FOR K2:=0 TO 5 DO
	 Cn_date[20,K2]:=0;
	 Cn_date[21,K2]:=0;
	 Cn_date[22,K2]:=0;
	 Cn_date[23,K2]:=0;
	 Cn_date[0,K2]:=0;
	 Cn_date[1,K2]:=0;
	 Cn_date[2,K2]:=0;
	 Cn_date[3,K2]:=0;
	 Cn_date[4,K2]:=0;
	 Cn_date[5,K2]:=0;
	 Cn_date[6,K2]:=0;
	 Cn_date[7,K2]:=0;
END_FOR
NGMark2[0,0]:=0;
NGMark2[1,0]:=0;
NGMark2[2,0]:=0;
NGMark2[3,0]:=0;
NGMark2[4,0]:=0;
NGMark2[5,0]:=0;
NGMark2[6,0]:=0;
NGMark2[7,0]:=0;
NGMark2[8,0]:=0;
NGMark2[9,0]:=0;
NGMark2[10,0]:=0;
NGMark2[11,0]:=0;
NGMark2[12,0]:=0;
NGMark2[13,0]:=0;
NGMark2[14,0]:=0;
NGMark2[0,0]:=0;
NGMark2[1,1]:=0;
NGMark2[2,1]:=0;
NGMark2[3,1]:=0;
NGMark2[4,1]:=0;
NGMark2[5,1]:=0;
NGMark2[6,1]:=0;
NGMark2[7,1]:=0;
NGMark2[8,1]:=0;
NGMark2[9,1]:=0;
NGMark2[10,1]:=0;
NGMark2[11,1]:=0;
NGMark2[12,1]:=0;
NGMark2[13,1]:=0;
NGMark2[14,1]:=0;
END_IF

END_FUNCTION_BLOCK

// ---- POUs/BasicFunction/Data/FB_DataTime.TcPOU
FUNCTION_BLOCK FB_DataTime
VAR_INPUT
	Month:INT;//实时月；
	dDay:INT;//实时日期；
	Hour:INT;//当前时间小时；
	Mins:INT;//分钟；
   Second:INT;//秒
    Alm :    BOOL ;//报警
	Wait :BOOL ;//待机
	Run :BOOL ;//运行
	JP_Wait:BOOL ;//极片更换时间
	Query:BOOL;//时间查询
	

END_VAR
VAR_OUTPUT
		STTimedata:ARRAY[0..32] OF ST_Timedata_2;

END_VAR
VAR
	
	rRun : R_TRIG;
	rAlm : R_TRIG;
	rWait : R_TRIG;
	rXL_Wait : R_TRIG;
	
	fRun: F_TRIG;
	fAlm: F_TRIG;
	fWait: F_TRIG;
    delay:BOOL ;//延时
	TON_1: TON;
	i:INT;
	K: INT;
	J: BOOL;
END_VAR

VAR_IN_OUT
     date1:INT;//查询日期
END_VAR

K:=K+1;
	IF K>499THEN
		J:=TRUE;
		K:=0;
	ELSE
		J:=FALSE;
	END_IF




///////////////运行时间/////////////////
rRun(CLK:= J , Q=> );

IF rRun.Q  AND  Run THEN
	STTimedata[System.StTime.wDay].RunTime[System.StTime.wHour]:=STTimedata[System.StTime.wDay].RunTime[System.StTime.wHour]+1;
END_IF

IF STTimedata[System.StTime.wDay].RunTime[System.StTime.wHour]> 3600 THEN
	STTimedata[System.StTime.wDay].RunTime[System.StTime.wHour]:= 3600 ;
END_IF

//IF STTimedata[System.StTime.wDay].AlmTime[System.StTime.wHour]= 0 AND STTimedata[System.StTime.wDay].WaitTime[System.StTime.wHour]= 0  AND 
 //   (STTimedata[System.StTime.wDay].RunTime[System.StTime.wHour]= 3585  OR  STTimedata[System.StTime.wDay].RunTime[System.StTime.wHour]= 3586 ) THEN
	//STTimedata[System.StTime.wDay].RunTime[System.StTime.wHour]:= 3600 ;
//END_IF


///////////////待机时间///////////////
rWait(CLK:=J , Q=> );

IF rWait.Q  AND Wait THEN
	STTimedata[System.StTime.wDay].WaitTime[System.StTime.wHour]:=STTimedata[System.StTime.wDay].WaitTime[System.StTime.wHour]+1;
END_IF

IF STTimedata[System.StTime.wDay].WaitTime[System.StTime.wHour]> 3600 THEN
	STTimedata[System.StTime.wDay].WaitTime[System.StTime.wHour]:= 3600 ;
END_IF

//IF STTimedata[System.StTime.wDay].RunTime[System.StTime.wHour]= 0 AND STTimedata[System.StTime.wDay].AlmTime[System.StTime.wHour]= 0  AND 
  //   (STTimedata[System.StTime.wDay].RunTime[System.StTime.wHour]= 3585  OR  STTimedata[System.StTime.wDay].RunTime[System.StTime.wHour]= 3586 )  THEN
//	STTimedata[System.StTime.wDay].WaitTime[System.StTime.wHour]:= 3600 ;
//END_IF


////////////////报警时间///////////////
rAlm(CLK:=J , Q=> );

IF rAlm.Q AND Alm THEN
	STTimedata[System.StTime.wDay].AlmTime[System.StTime.wHour]:=STTimedata[System.StTime.wDay].AlmTime[System.StTime.wHour]+1;
END_IF

IF STTimedata[System.StTime.wDay].AlmTime[System.StTime.wHour]> 3600 THEN
	STTimedata[System.StTime.wDay].AlmTime[System.StTime.wHour]:= 3600 ;
END_IF

//IF STTimedata[System.StTime.wDay].RunTime[System.StTime.wHour]= 0 AND STTimedata[System.StTime.wDay].WaitTime[System.StTime.wHour]= 0  AND
//    (STTimedata[System.StTime.wDay].RunTime[System.StTime.wHour]= 3585  OR  STTimedata[System.StTime.wDay].RunTime[System.StTime.wHour]= 3586 ) THEN
//	STTimedata[System.StTime.wDay].AlmTime[System.StTime.wHour]:= 3600 ;
//END_IF

////////////////下料等待托盘时间///////////////
rXL_Wait(CLK:=J, Q=> );

IF rXL_Wait.Q AND JP_Wait THEN
	STTimedata[System.StTime.wDay].changeTime[System.StTime.wHour]:=STTimedata[System.StTime.wDay].changeTime[System.StTime.wHour]+1;
END_IF

//数据查询
IF Query THEN
	delay:=TRUE;
END_IF

TON_1(IN:= , PT:=T#60S , Q=> , ET=> );
IF delay THEN
		  IF NOT TON_1.Q THEN
			  TON_1.IN:=TRUE;
		  ELSE	
			  delay:=FALSE;
			  date1:=System.StTime.wDay;
		  END_IF	 
ELSE	
	 TON_1.IN:=FALSE;
END_IF


IF NOT delay THEN
STTimedata[32]:=STTimedata[System.StTime.wDay];
ELSE
STTimedata[32]:=STTimedata[date1];
END_IF

//数据清零
IF (System.StTime.wMonth=2 AND  System.StTime.wDay=28 )   OR
    ((System.StTime.wMonth=4 OR System.StTime.wMonth=6 OR System.StTime.wMonth=9 OR System.StTime.wMonth=11) AND System.StTime.wDay=30 )   OR
	((System.StTime.wMonth=1 OR  System.StTime.wMonth=3 OR System.StTime.wMonth=5 OR System.StTime.wMonth=7 OR System.StTime.wMonth=8 OR System.StTime.wMonth=10 OR System.StTime.wMonth=12) AND  System.StTime.wDay=31)  AND
    System.StTime.wHour=23 AND   System.StTime.wMinute =59 AND  System.StTime.wSecond =59 THEN
	FOR i:=0 TO 32  DO
	MEMSET(ADR(STTimedata[i]),0,SIZEOF(STTimedata[i]));	
	END_FOR
END_IF

END_FUNCTION_BLOCK

// ---- POUs/BasicFunction/Data/CS_Recipe.TcPOU
FUNCTION_BLOCK CS_Recipe
VAR_INPUT
END_VAR
VAR_OUTPUT
END_VAR
VAR
	


 //recipeManCommands: RecipeManCommands;
	result: DWORD;
END_VAR

VAR_IN_OUT
  iRecipe2:    IRecipe;
END_VAR





(*

IF iRecipe2.bCreate THEN
   result:= recipeManCommands.CreateRecipe(RecipeDefinitionName:='Recipes' , RecipeName:='SJ_Rec' );
   iRecipe2.bCreate:=FALSE;
END_IF

IF iRecipe2.bSave THEN
    result:= recipeManCommands.ReadAndSaveRecipeAs(RecipeDefinitionName:='Recipes' , RecipeName:='SJ_Rec' , FileName:='C:\P2Data\P2Par');
    iRecipe2.bSave:=FALSE;
END_IF

IF iRecipe2.bLoad THEN
	result:= RecipeManCommands.LoadFromAndWriteRecipe(RecipeDefinitionName:='Recipes' , RecipeName:='SJ_Rec' , FileName:='C:\P2Data\P2Par');
    iRecipe2.bLoad:=FALSE;
END_IF

*)

END_FUNCTION_BLOCK

// ---- POUs/BasicFunction/MES/CS_CcdTcp_V2.TcPOU
FUNCTION_BLOCK PUBLIC CS_CcdTcp_V2
VAR_INPUT
END_VAR
VAR_OUTPUT
END_VAR
VAR_IN_OUT
   iCcd2:ST_CCDCom;
   Data:STCcdData;
END_VAR


VAR
	ccdDataSend:STCcdDataSend;
	ccdDataReceive:STCcdDataSend;
	fbTcpCon:FB_SocketConnect;
	fbTcpSend:FB_SocketSend;
	fbTcpRec:FB_SocketReceive;
	fbTcpClose: FB_SocketClose;
	bConnect: BOOL;
	bClose: BOOL;
	hTcpSock: T_HSOCKET;
	//aTcpSend:ARRAY[1..10] OF BYTE;
	//aTcpReceive:ARRAY[1..10] OF BYTE;	
	StrSend:STRING;
	StrReceive:STRING;
	fbUdpCreate:FB_SocketUdpCreate;
	hUdp: T_HSOCKET;
	bCreate: BOOL;
	port: UDINT:=9004;
	bSendTcp: BOOL;
	bReceiveTcp: BOOL;
	fbSwingHalt2: MC_Halt;

    strReceiveData: STCcdData;

	iorderTemp: DINT;
	TON100:TON;
END_VAR




	Config();
	
	M_SendReceive();


	
	

	
	
	
	

	
	
	
	
	
	
	
	
	
	
	
	
	
	
	
	
	
(*	
   fbUdpCreate(
	sSrvNetId:= , 
	sLocalHost:= , 
	nLocalPort:= port, 
	bExecute:=bCreate , 
	tTimeout:= , 
	bBusy=> , 
	bError=> , 
	nErrId=> , 
	hSocket=> hUdp);
	
	
	*)

ACTION Config:



  IF iCcd2.bComOpen THEN
	 bConnect:=TRUE;	
	 bClose:=FALSE;
	 iCcd2.bComOpen:=FALSE;
  END_IF
  
   IF iCcd2.bComClose THEN
	 bConnect:=FALSE;	
	 bClose:=TRUE;
	 iCcd2.bComClose:=FALSE;
  END_IF 
  
  
  
fbTcpCon(
	sSrvNetId:= ''   ,          //       (*'169.254.46.193.1.1'*) , 
	sRemoteHost:='192.168.2.11'     , 
	nRemotePort:= 2020, 
	bExecute:=bConnect , 
	tTimeout:= , 
	bBusy=> , 
	bError=> , 
	nErrId=> , 
	hSocket=>hTcpSock );
	
fbTcpClose(
	sSrvNetId:= ''   , 
	hSocket:=hTcpSock , 
	bExecute:=bClose , 
	tTimeout:=T#5S , 
	bBusy=> , 
	bError=> , 
	nErrId=> );


IF fbTcpCon.bBusy THEN
	bConnect:=FALSE;
END_IF

IF fbTcpClose.bBusy THEN
   bClose:=FALSE;
END_IF
END_ACTION

ACTION M_SendReceive:



  IF iCcd2.bSend THEN
	 bSendTcp:=TRUE;
	 iCcd2.bDone:=FALSE;
	 iCcd2.bError:=FALSE;
	 //iCcd2.strReceive:='';
    MEMSET(ADR(ccdDataSend.strBetryName),0,SIZEOF(ccdDataSend.strBetryName));
	MEMSET(ADR(ccdDataSend.strCode),0,SIZEOF(ccdDataSend.strCode));
	MEMSET(ADR(ccdDataSend.strShortData),0,SIZEOF(ccdDataSend.strShortData));
	MEMSET(ADR(ccdDataSend.strHotPress),0,SIZEOF(ccdDataSend.strHotPress));
    STRING_TO_UTF8(pDstUTF8:=ADR(ccdDataSend.strBetryName) , pSrcSTRING:=ADR(Data.strBetryName) , nDstSize:=INT_TO_UINT( LEN(STR:=Data.strBetryName )+1) );
    STRING_TO_UTF8(pDstUTF8:=ADR(ccdDataSend.strCode) , pSrcSTRING:=ADR(Data.strCode) , nDstSize:=INT_TO_UINT( LEN(STR:=Data.strCode )+1) ); 
    STRING_TO_UTF8(pDstUTF8:=ADR(ccdDataSend.strShortData) , pSrcSTRING:=ADR(Data.strShortData) , nDstSize:=INT_TO_UINT( LEN(STR:=Data.strShortData )+1) );
	STRING_TO_UTF8(pDstUTF8:=ADR(ccdDataSend.strHotPress) , pSrcSTRING:=ADR(Data.strHotPress) , nDstSize:=INT_TO_UINT( LEN(STR:=Data.strHotPress )+1) );
    iCcd2.bSend:=FALSE;
	iorderTemp:=Data.iorder;
	TON100.IN:=TRUE;
END_IF
	 
fbTcpSend(
		sSrvNetId:= , 
		hSocket:=hTcpSock , 
		cbLen:=SIZEOF(ccdDataSend), 
		pSrc:= ADR(ccdDataSend), 
		bExecute:= bSendTcp, 
		tTimeout:= T#2S , 
		bBusy=> , 
		bError=> , 
		nErrId=> );
	IF bSendTcp AND fbTcpSend.bBusy THEN
		bSendTcp:=FALSE;
	END_IF
	
	
bReceiveTcp:=NOT bReceiveTcp;
	
fbTcpRec(
	sSrvNetId:= , 
	hSocket:= hTcpSock, 
	cbLen:=SIZEOF(ccdDataReceive) , 
	pDest:=ADR(ccdDataReceive) , 
	bExecute:=bReceiveTcp , 
	tTimeout:= T#5S, 
	bBusy=> , 
	bError=> , 
	nErrId=> , 
	nRecBytes=> );

	
TON100(IN:= , PT:= T#3S, Q=> , ET=> );//通讯超时
	
 ccdDataReceive.iorder;	//功能码 2     3      4
 UTF8_TO_STRING (pDstSTRING:= ADR(strReceiveData.strBetryName) , pSrcUTF8:= ADR(ccdDataReceive.strBetryName), nDstSize:=SIZEOF(ccdDataReceive.strBetryName) , nDstLen=> );//文件名

	IF ccdDataReceive.iorder=iorderTemp  AND ccdDataReceive.iorder>0  THEN  //发送对应 返回功能码  
		
        IF ccdDataReceive.iorder=2 THEN     //给MES发送数据成功
		    iCcd2.bDone:=TRUE; 
		ELSIF ccdDataReceive.iorder=3 THEN   //取料请求文件名成功  有可能文件名是空
			IF strReceiveData.strBetryName='' THEN //文件名空  给plc自定义文件名   也可以做报警    
			   iCcd2.bDone:=TRUE; 
			    iCcd2.strReceive:= MAIN.strTime;
			ELSE
			 iCcd2.strReceive:= strReceiveData.strBetryName;
			  iCcd2.bDone:=TRUE; 
			END_IF
		ELSIF ccdDataReceive.iorder=4 THEN   //取料夹爪夹空   不用处理文件名字
		    iCcd2.bDone:=TRUE; 
			iCcd2.strReceive:='';
		END_IF
	
	   MEMSET(ADR(ccdDataReceive),0,SIZEOF(ccdDataReceive));
	   iorderTemp:=0;
	   TON100.IN:=FALSE;
	END_IF
	
	IF TON100.Q AND iorderTemp<>0 THEN  //通讯超时报警
		   ;           //报警信号
		 TON100.IN:=FALSE;
		  iorderTemp:=0;
	END_IF
END_ACTION

END_FUNCTION_BLOCK

// ---- POUs/BasicFunction/Basic/07_Ten/FB_TensionPole.TcPOU
FUNCTION_BLOCK FB_TensionPole  //只和Tim轴联动    学习放卷与摆杆的角度即可   张力使能直接开

VAR_INPUT
	bReset			           :BOOL;	 //复位       
	bCcw		                   :BOOL;	//放卷电机方向选择    
    fDanserDegree         :REAL;//摆杆实时位置
  
    fActTorque               :REAL; //当前力矩值
    fSetTorque               :REAL; //设定力矩值
	
    PidSwitch                    :BOOL;	   //PID功能选择
   

   	fStudyDiameter          :REAL;  //摆杆学习时放卷轴卷径   人工HMI输入
	
	fDriveDiameter	        :REAL:=80;//驱动实轴直径	计算卷径时使用
    fPoleWith                   :REAL;//片宽     下个周期主驱补偿，片宽变化，放卷也应相应变化才对。
 	fCompensation                          :REAL;//主驱补偿值
	fDancerMinPos	:REAL;	//摆杆最小值
	fDancerMaxPos	:REAL;	//摆杆最大值
	fDanceBlancePos	:REAL;	//摆杆平衡值
	bStudyExecute                      :BOOL;       //摆杆学习使能	
END_VAR

VAR_OUTPUT
	bReady                 :BOOL;  
	bTensionOK		 	:BOOL;	

	bError			   	:BOOL;		                          
END_VAR


VAR_IN_OUT
	VirMain         :axis_ref;	//虚拟主轴	   
	Master	     	:axis_ref;	//驱动放卷虚拟轴	   
    Slave		        :axis_ref;  //放卷实轴
	Driver		    :axis_ref; //驱动实轴
	TimerAxis	    :axis_ref;	// 摆杆张力放卷虚拟轴  
	TensionAxis   :axis_ref;  //张力轴

   	bTenExecute		        :BOOL;	//张力使能
	Table		    :ARRAY[0..105,1..2]OF REAL;	
END_VAR

VAR
	iFlgwind :INT;
    fWindDiameter         :REAL;//放卷轴实时卷径AI
	
	
	
	bAxisError:BOOL;
	rtEnable		:R_TRIG;  
	ftEnable		:F_TRIG;

	TON02: TON;
	
	rTRIG100: R_TRIG;
	iTensionStep:UINT;
	fCcw: REAL;	(*选择放卷方向后*)
	fbGearOut						:MC_GearOut;		//Unwind

	fRatio1: LREAL;
	fRatio2: LREAL;

	fbJogUnwind: MC_Jog;    //Unwind

	fKp2: LREAL;(*乘数系数*)
	Ti: LREAL;
	fbHalt: MC_Halt; // Unwind
    fbHaltTensionAxis: MC_Halt; // Unwind        
	
	
	bPosLimitError			:BOOL;		
	bNegLimitError			:BOOL;		
	bTorqueError			:BOOL;	
	bTenOKTimeError			:BOOL;
	
	fCalcDancerPos1: REAL;
	fCalcDancerPos2: REAL;


	Delay1,Delay2: TON;
	Delay3:            TON;
	Delay4:            TON;
	rtStudy	   :R_TRIG;
	ftStudy	   :F_TRIG;


	bStudyFinish: BOOL; 
	studyStage: INT;
	ad_Set_test: REAL;
	struckstudying: BOOL;
	structTime: INT;
	// 学习计数
	structPrinter: INT;
	structAcc: REAL;
	structAxisPosPast: LREAL;
	structAxisPosNow: LREAL;
	gear: REAL := 1;
	iwindJog: INT;// 1收卷  2放卷 3停止

	DA1: REAL;
	DA2: INT;
	DA3: INT;

	bFunBlokError: BOOL;

	fMasterLinerSpeed: REAL;
	TM: REAL:=1;
	TM_old: REAL;
	fbGearDync :MC_GearInMultiMaster;
	iFlgStart: INT;

	DelayDiaMeter:TON;
	RDiaMeter  :R_TRIG;
	RDiaMeter2  :R_TRIG;
    tonDiaMeter  :Tc2_Standard.TON;

	_fUwPos1,_fUwPos2,_fUwPos3	:LREAL;
	_fDancerPos1,_fDancerPos2,_fDancerPos3	:LREAL;
	_fDrivePos1,_fDrivePos2,_fDrivePos3	:LREAL;
    iUnwindStartPos: LREAL;
	iUnwindOldTurns: DINT;
	fDeltaUwPos1,_fDeltaUwPos1	:LREAL;
	fDeltaDrivePos1,_fDeltaDrivePos1	:LREAL;
	fDeltaDancerPos1,_fDeltaDancerPos1:LREAL;
	iUnwindStartTurns: DINT;


	fDiameterCalculate: LREAL;//放卷轴采样卷径
	fWindDiameterTemp: REAL;//放卷轴卷径-采用
	fWindFirstPos: LREAL;
	fWindLengh: LREAL;
	rtrigs		:ARRAY[1..3]OF R_TRIG;
	fFlgCalculateOnce: BOOL;
	fPos1Length: REAL;
	fPos2Length: REAL;
	fWindPos1Deg: REAL;
	fWindPos2Deg: REAL;
	fDanceBlancePosTemp: REAL;
	bFlgDiameterCalculate: BOOL;
END_VAR



TON02(IN:= , PT:=T#10MS , Q=> , ET=> );

Study();
fCcw:=SEL(bCcw,1,-1);	

//fCalcDancerPos1:=0.75*fDancerMinPos+0.25*fDanceBlancePos;	
fCalcDancerPos1:=fDancerMinPos+5;	
//fCalcDancerPos2:=0.75*fDancerMaxPos+0.25*fDanceBlancePos;	
//fCalcDancerPos2:=0.65*fDancerMaxPos+0.25*fDanceBlancePos;	
fCalcDancerPos2:=fDancerMaxPos-20;
rtEnable(CLK:=bTenExecute , Q=> );        
ftEnable(CLK:=bTenExecute , Q=> );    
rtrigs	[1](CLK:=VirMain.Status.Moving AND  VirMain.NcToPlc.ModuloActPos>=355 AND VirMain.NcToPlc.ModuloActPos<360 OR rtEnable.Q AND VirMain.Status.NotMoving , Q=> ); 

bReady:= NOT bAxisError  AND NOT bError AND  iTensionStep=1 AND NOT bFunBlokError  
               AND Master.Status.NotMoving AND TimerAxis.Status.Moving  AND NOT Slave.Status.Coupled  AND Slave.Status.NotMoving
               AND Master.Status.ControlLoopClosed AND TimerAxis.Status.ControlLoopClosed   AND Slave.Status.ControlLoopClosed  AND 
               TimerAxis.Status.ConstantVelocity  AND 
                 ABS(fActTorque -fSetTorque )<10   ;
 
 fWindDiameter:= LIMIT(250,fWindDiameter,800);  //模糊卷径
				 			 
CASE iTensionStep OF
0:
    fbJogUnwind.Velocity:=15;
    fbGearDync.Enable:=FALSE;
	fbGearOut.Execute:=FALSE;
	fbHalt.Execute:=FALSE;
   fbHaltTensionAxis.Execute:=FALSE;    //停止张力轴
    iwindJog:=3;
	bTensionOK:=FALSE;
	TON02.IN:=FALSE;
    iTensionStep:=1;  
1:
  IF bTenExecute AND bReady THEN
    	iTensionStep:=120;  
  END_IF
  IF ftEnable.Q THEN
    	iTensionStep:=630; 
  END_IF
 
120:  //低位
     TM:=3;
	 fPos1Length:=0;
	 fPos2Length:=0;	 
	 fWindPos1Deg:=0;
	 fWindPos2Deg:=0;
     fDanceBlancePosTemp:=fCalcDancerPos1;
	 iTensionStep:=130;  		
130:  	
	 fbGearDync.Enable:=TRUE;    //开启耦合
     fWindFirstPos:=Slave.NcToPlc.ActPos;
	 iTensionStep:=140;  
140:  
	IF  Slave.Status.Coupled  AND bTenExecute AND NOT fbGearDync.Error AND NOT fbGearDync.CommandAborted   AND NOT bTenOKTimeError AND NOT  bTorqueError THEN
		IF   (fDanserDegree<fCalcDancerPos1+6  AND fDanserDegree>fCalcDancerPos1-6)     THEN
		     fPos1Length:=f_Length2(Table:=Table,X:=fDanserDegree);
			 fWindPos1Deg:=Slave.NcToPlc.ActPos;
		     iTensionStep:=200;
		END_IF	
	ELSIF fbGearDync.Error OR fbGearDync.CommandAborted   OR bTenOKTimeError OR  bTorqueError OR NOT bTenExecute     THEN
		  iTensionStep:=630;
	END_IF

      fWindLengh:= ABS( FC_AngleToLength(Slave.NcToPlc.ActPos,fWindDiameterTemp)- FC_AngleToLength(fWindFirstPos,fWindDiameterTemp) );
      IF fWindLengh>800 THEN
          bError:=TRUE;
          iTensionStep:=630;
     END_IF	 
	 
	 
	 
	200: 
	      fDanceBlancePosTemp:=fCalcDancerPos2;
	       iTensionStep:=210;  		
	210: 	 
	 IF  Slave.Status.Coupled  AND bTenExecute AND NOT fbGearDync.Error AND NOT fbGearDync.CommandAborted   AND NOT bTenOKTimeError AND NOT  bTorqueError THEN
		IF   (fDanserDegree<fCalcDancerPos2+6  AND fDanserDegree>fCalcDancerPos2-6)     THEN
		     fPos2Length:=f_Length2(Table:=Table,X:=fDanserDegree);
			 fWindPos2Deg:=Slave.NcToPlc.ActPos;
		     iTensionStep:=300;
		END_IF	
	ELSIF fbGearDync.Error OR fbGearDync.CommandAborted   OR bTenOKTimeError OR  bTorqueError OR NOT bTenExecute     THEN
		  iTensionStep:=630;
	END_IF
	 
	   fWindLengh:= ABS( FC_AngleToLength(Slave.NcToPlc.ActPos,fWindDiameterTemp)- FC_AngleToLength(fWindFirstPos,fWindDiameterTemp) );
      IF fWindLengh>800 THEN
          bError:=TRUE;
          iTensionStep:=630;
     END_IF	 
	 
 300:
       fWindDiameter:= ABS(   (fPos2Length-fPos1Length)*360 /  ( (fWindPos2Deg-fWindPos1Deg)*Tc2_System.PI )  ) ;
	 	fDanceBlancePosTemp:=fDanceBlancePos;
		 TM:=1;
	    iTensionStep:=550;  		
	 
550:

	IF  Slave.Status.Coupled  AND bTenExecute AND NOT fbGearDync.Error AND NOT fbGearDync.CommandAborted   AND NOT bTenOKTimeError AND NOT  bTorqueError THEN
		IF   (fDanserDegree<fDanceBlancePos+5  AND fDanserDegree>fDanceBlancePos-5)  AND PidSwitch   THEN
			bTensionOK:=TRUE;
			iTensionStep:=600;
        ELSIF NOT PidSwitch THEN
			bTensionOK:=TRUE;
			iTensionStep:=600;
		END_IF
	ELSIF fbGearDync.Error OR fbGearDync.CommandAborted   OR bTenOKTimeError OR  bTorqueError OR NOT bTenExecute     THEN
		  iTensionStep:=630;
	END_IF

	
      fWindLengh:= ABS( FC_AngleToLength(Slave.NcToPlc.ActPos,fWindDiameterTemp)- FC_AngleToLength(fWindFirstPos,fWindDiameterTemp) );
      IF fWindLengh>800 THEN
          bError:=TRUE;
          iTensionStep:=630;
     END_IF

(******************************  进入平衡运行阶段   *************************************)
600:
	IF ( bPosLimitError OR bNegLimitError OR  bTorqueError   OR bTenOKTimeError OR   (NOT bTenExecute)  OR bAxisError 
        OR TimerAxis.Status.NotMoving  ) AND PidSwitch     THEN  
	    TON02.IN:=TRUE;
    ELSIF  ( NOT bTenExecute  OR bAxisError  ) AND  NOT  PidSwitch     THEN 
       TON02.IN:=TRUE;
	END_IF
	
	IF TON02.Q THEN   
		IF ( bPosLimitError  OR bNegLimitError OR  bTorqueError  OR  bAxisError OR bFunBlokError OR bTenOKTimeError ) AND   PidSwitch   THEN
		   bError:=TRUE;
       ELSIF   (  bAxisError OR bFunBlokError  ) AND  NOT  PidSwitch     THEN
            bError:=TRUE;
		END_IF
	    iTensionStep:=630;
	    TON02.IN:=FALSE; 	
	END_IF
	
(******************************  解耦*************************************)
630:
     fbGearDync.Enable:=FALSE;    //开启耦合
	 bTenExecute:=FALSE;
     iTensionStep:=640;	
640:
     IF   NOT  fbGearDync.InGear  THEN
         iTensionStep:=650;	
     END_IF
650:
	IF Slave.Status.Coupled THEN
		fbGearOut.Execute:=TRUE;
		iTensionStep:=700;
	ELSE
		iTensionStep:=700;	
	END_IF
700:
	IF NOT Slave.Status.Coupled   THEN
        fbGearOut.Execute:=FALSE;
		bTensionOK:=FALSE;
		bFlgDiameterCalculate:=FALSE;
		fbHalt.Execute:=TRUE;   
		iTensionStep:=750;	
	END_IF
750:
	IF Slave.Status.NotMoving  THEN  
	   iTensionStep:=800;  //0
	END_IF		

800:
  IF NOT bTorqueError THEN  
	      iTensionStep:=0;  
 ELSE
	    fbHaltTensionAxis.Execute:=FALSE;    //停止张力轴
		 iTensionStep:=810;  //0
  END_IF
810:
       iTensionStep:=0;  //0
END_CASE

(*********************************** 耦合  *********************************************)
  // TM:=0.012*ABS(  f_Length2(Table:=Table,X:=fDanserDegree)-f_Length2(Table:=Table,X:=fDanceBlancePos))+0.4;
  
      IF  NOT  bFlgDiameterCalculate   THEN    //ABS(fWindDiameter-fDiameterCalculate)>=25
           fWindDiameterTemp:=fWindDiameter;
      ELSE
          fWindDiameterTemp:=fDiameterCalculate;
     END_IF

 // fWindDiameterTemp:=fWindDiameter;

//fRatio1:=fCcw*fDriveDiameter/fWindDiameterTemp;
IF fWindDiameterTemp<>0 THEN
	IF rtrigs	[1].Q THEN
		fRatio1:=fCcw*(fPoleWith+fCompensation)/(fWindDiameterTemp*Tc2_System.PI);     
	END_IF                   
	Ti:=1;
		fKp2:=(( f_Length2(Table:=Table,X:=fDanserDegree)-f_Length2(Table:=Table,X:=fDanceBlancePosTemp) )*360 ) / (Tc2_System.PI*fWindDiameterTemp*100*TM);
	IF ABS(fKp2)>0.005 THEN		
		fRatio2:=SEL(PidSwitch,0, fCcw*fKp2) ;
	ELSE
		fRatio2:=SEL(PidSwitch,0, 0) ;
	END_IF
END_IF

(********************************* 初始卷 后 循环更新半径  *********************************************)
DelayDiaMeter(IN:= bTensionOK, PT:=T#2S , Q=> , ET=> );
RDiaMeter(CLK:=DelayDiaMeter.Q , Q=> );
IF RDiaMeter.Q THEN
	_fDrivePos1:=Driver.NcToPlc.ActPos;		//驱动辊位置锁存
	_fUwPos1:=   Slave.NcToPlc.ActPos;        //放卷位置所存
   _fDancerPos1:=fDanserDegree;              //摆杆位置锁存

   iUnwindStartPos:= Slave.NcToPlc.ActPos;
   iUnwindOldTurns:=10;
END_IF

	IF  DelayDiaMeter.Q THEN  
        iUnwindStartTurns:=  ABS(  LREAL_TO_DINT ( (  FC_AngleToLength( Driver.NcToPlc.ActPos,fDriveDiameter)  - FC_AngleToLength( _fDrivePos1,fDriveDiameter) )/100 )  ) ;  
        //tonDiaMeter(IN:= ABS( Driver.NcToPlc.SetVelo)<0.2 , PT:=T#100MS , Q=> , ET=> );

		IF iUnwindStartTurns>=iUnwindOldTurns  AND  VirMain.NcToPlc.ModuloSetPos>=352   AND  VirMain.NcToPlc.ModuloSetPos<=360  THEN  //   计算一次卷径
			_fDeltaDrivePos1:=ABS(Driver.NcToPlc.ActPos-_fDrivePos1);
			_fDeltaUwPos1:=ABS(Slave.NcToPlc.ActPos-_fUwPos1);
			_fDeltaDancerPos1:=fDanserDegree;
            DA1:=     f_Length2(Table:=Table,X:=_fDeltaDancerPos1)-f_Length2(Table:=Table,X:=_fDancerPos1) ;
			IF _fDeltaUwPos1<>0 THEN
          			 fDiameterCalculate:= ( FC_AngleToLength(_fDeltaDrivePos1,fDriveDiameter)- ( f_Length2(Table:=Table,X:=_fDeltaDancerPos1)-f_Length2(Table:=Table,X:=_fDancerPos1))  ) *360/ (PI*_fDeltaUwPos1) ;
		   	END_IF
            // fDiameterCalculate:= ( FC_AngleToLength(_fDeltaDrivePos1,fDriveDiameter)  ) *360/ (PI*_fDeltaUwPos1) ;
			_fDrivePos1:=Driver.NcToPlc.ActPos;		
			_fUwPos1:=Slave.NcToPlc.ActPos;
			_fDancerPos1:=fDanserDegree;
			iUnwindOldTurns:=10;
			bFlgDiameterCalculate:=TRUE;
		END_IF
		
	END_IF


(***********************************错误报警*********************************************)	
bAxisError:=      Slave.Status.Error OR  Master.Status.Error OR  TimerAxis.Status.Error ;
bFunBlokError:=fbGearDync.Error OR fbGearOut.Error OR fbHalt.Error OR fbJogUnwind.Error  ;
			
IF  bReset AND iTensionStep<>600  AND bError   THEN   //复位处理
    bError:=FALSE;
	iTensionStep:=630;
END_IF

(************************************  张力出错和取消的处理  ******************************************************)
Delay1(IN:=fDanserDegree>fDancerMaxPos AND bTensionOK , PT:=T#300MS , Q=> , ET=> );
bPosLimitError:=Delay1.Q;
Delay2(IN:=fDanserDegree<fDancerMinPos AND bTensionOK , PT:=T#300MS , Q=> , ET=> );
bNegLimitError:=Delay2.Q;
Delay3(IN:=( ABS(fActTorque -fSetTorque )>=10 OR  fDanserDegree> fDancerMaxPos+35 OR  fDanserDegree< fDancerMinPos-35)   AND   bTensionOK , PT:=T#300MS , Q=> , ET=> );
bTorqueError:=Delay3.Q;
Delay4(IN:=( iTensionStep=550 OR  iTensionStep=600 ) AND  Master.Status.NotMoving   AND (fDanserDegree>fDanceBlancePos+20  OR fDanserDegree<fDanceBlancePos-20)  AND ABS(fRatio2)>0.005 AND PidSwitch , PT:=T#5S , Q=> , ET=> );
bTenOKTimeError:=Delay4.Q;

Jog();
Motion();
TM_old:=TM;






(*
TON02(IN:= , PT:=T#10MS , Q=> , ET=> );

Study();
fCcw:=SEL(bCcw,1,-1);	

fCalcDancerPos1:=0.75*fDancerMinPos+0.25*fDanceBlancePos;	
fCalcDancerPos2:=0.75*fDancerMaxPos+0.25*fDanceBlancePos;	

rtEnable(CLK:=bTenExecute , Q=> );        
ftEnable(CLK:=bTenExecute , Q=> );    
rtrigs	[1](CLK:=VirMain.Status.Moving AND  VirMain.NcToPlc.ModuloActPos>=355 AND VirMain.NcToPlc.ModuloActPos<360 OR rtEnable.Q AND VirMain.Status.NotMoving , Q=> ); 

bReady:= NOT bAxisError  AND NOT bError AND  iTensionStep=1 AND NOT bFunBlokError  
               AND Master.Status.NotMoving AND TimerAxis.Status.Moving  AND NOT Slave.Status.Coupled  AND Slave.Status.NotMoving
               AND Master.Status.ControlLoopClosed AND TimerAxis.Status.ControlLoopClosed   AND Slave.Status.ControlLoopClosed  AND 
               TimerAxis.Status.ConstantVelocity  AND 
                 ABS(fActTorque -fSetTorque )<10   ;
 
CASE iTensionStep OF
0:
    fbJogUnwind.Velocity:=15;
    fbGearDync.Enable:=FALSE;
	fbGearOut.Execute:=FALSE;
	fbHalt.Execute:=FALSE;
   fbHaltTensionAxis.Execute:=FALSE;    //停止张力轴
    iwindJog:=3;
	bTensionOK:=FALSE;
	TON02.IN:=FALSE;
    iTensionStep:=1;  
1:
  IF bTenExecute AND bReady THEN
    	iTensionStep:=120;  
  END_IF
  IF ftEnable.Q THEN
    	iTensionStep:=630; 
  END_IF
 
120:  
	 fbGearDync.Enable:=TRUE;    //开启耦合
     fWindFirstPos:=Slave.NcToPlc.ActPos;
	 iTensionStep:=550;  
550:

	IF  Slave.Status.Coupled  AND bTenExecute AND NOT fbGearDync.Error AND NOT fbGearDync.CommandAborted   AND NOT bTenOKTimeError AND NOT  bTorqueError THEN
		IF   (fDanserDegree<fDanceBlancePos+5  AND fDanserDegree>fDanceBlancePos-5)  AND PidSwitch   THEN
			bTensionOK:=TRUE;
			iTensionStep:=600;
        ELSIF NOT PidSwitch THEN
			bTensionOK:=TRUE;
			iTensionStep:=600;
		END_IF
	ELSIF fbGearDync.Error OR fbGearDync.CommandAborted   OR bTenOKTimeError OR  bTorqueError OR NOT bTenExecute     THEN
		  iTensionStep:=630;
	END_IF

      fWindLengh:= ABS( FC_AngleToLength(Slave.NcToPlc.ActPos,fWindDiameterTemp)- FC_AngleToLength(fWindFirstPos,fWindDiameterTemp) );
      IF fWindLengh>800 THEN
          bError:=TRUE;
          iTensionStep:=630;
     END_IF

(******************************  进入平衡运行阶段   *************************************)
600:
	IF ( bPosLimitError OR bNegLimitError OR  bTorqueError   OR bTenOKTimeError OR   (NOT bTenExecute)  OR bAxisError 
        OR TimerAxis.Status.NotMoving  ) AND PidSwitch     THEN  
	    TON02.IN:=TRUE;
    ELSIF  ( NOT bTenExecute  OR bAxisError  ) AND  NOT  PidSwitch     THEN 
       TON02.IN:=TRUE;
	END_IF
	
	IF TON02.Q THEN   
		IF ( bPosLimitError  OR bNegLimitError OR  bTorqueError  OR  bAxisError OR bFunBlokError OR bTenOKTimeError ) AND   PidSwitch   THEN
		   bError:=TRUE;
       ELSIF   (  bAxisError OR bFunBlokError  ) AND  NOT  PidSwitch     THEN
            bError:=TRUE;
		END_IF
	    iTensionStep:=630;
	    TON02.IN:=FALSE; 	
	END_IF
	
(******************************  解耦*************************************)
630:
     fbGearDync.Enable:=FALSE;    //开启耦合
	 bTenExecute:=FALSE;
     iTensionStep:=640;	
640:
     IF   NOT  fbGearDync.InGear  THEN
         iTensionStep:=650;	
     END_IF
650:
	IF Slave.Status.Coupled THEN
		fbGearOut.Execute:=TRUE;
		iTensionStep:=700;
	ELSE
		iTensionStep:=700;	
	END_IF
700:
	IF NOT Slave.Status.Coupled   THEN
        fbGearOut.Execute:=FALSE;
		bTensionOK:=FALSE;
		fFlgCalculateOnce:=FALSE;
		fbHalt.Execute:=TRUE;   
		iTensionStep:=750;	
	END_IF
750:
	IF Slave.Status.NotMoving  THEN  
	   iTensionStep:=800;  //0
	END_IF		

800:
  IF NOT bTorqueError THEN  
	      iTensionStep:=0;  
 ELSE
	    fbHaltTensionAxis.Execute:=FALSE;    //停止张力轴
		 iTensionStep:=810;  //0
  END_IF
810:
       iTensionStep:=0;  //0
END_CASE

(*********************************** 耦合  *********************************************)
  // TM:=0.012*ABS(  f_Length2(Table:=Table,X:=fDanserDegree)-f_Length2(Table:=Table,X:=fDanceBlancePos))+0.4;
TM:=1;
      IF NOT fFlgCalculateOnce THEN  //        ABS(fWindDiameter-fDiameterCalculate)>=80
           fWindDiameterTemp:=fWindDiameter;
      ELSE
          fWindDiameterTemp:=fDiameterCalculate;
     END_IF

 // fWindDiameterTemp:=fWindDiameter;

//fRatio1:=fCcw*fDriveDiameter/fWindDiameterTemp;
IF fWindDiameterTemp<>0 THEN
	IF rtrigs	[1].Q THEN
		fRatio1:=fCcw*(fPoleWith+fCompensation)/(fWindDiameterTemp*Tc2_System.PI);     
	END_IF                   
	Ti:=1;
		fKp2:=(( f_Length2(Table:=Table,X:=fDanserDegree)-f_Length2(Table:=Table,X:=fDanceBlancePos) )*360 ) / (Tc2_System.PI*fWindDiameterTemp*100*TM);
	IF ABS(fKp2)>0.005 THEN		
		fRatio2:=SEL(PidSwitch,0, fCcw*fKp2) ;
	ELSE
		fRatio2:=SEL(PidSwitch,0, 0) ;
	END_IF
END_IF

(********************************* 初始卷 后 循环更新半径  *********************************************)
DelayDiaMeter(IN:= bTensionOK, PT:=T#2S , Q=> , ET=> );
RDiaMeter(CLK:=DelayDiaMeter.Q , Q=> );
IF RDiaMeter.Q THEN
	_fDrivePos1:=Driver.NcToPlc.ActPos;		//驱动辊位置锁存
	_fUwPos1:=   Slave.NcToPlc.ActPos;        //放卷位置所存
   _fDancerPos1:=fDanserDegree;              //摆杆位置锁存

   iUnwindStartPos:= Slave.NcToPlc.ActPos;
   iUnwindOldTurns:=10;
END_IF

	IF  DelayDiaMeter.Q THEN  
        iUnwindStartTurns:=  ABS(  LREAL_TO_DINT ( (  FC_AngleToLength( Driver.NcToPlc.ActPos,fDriveDiameter)  - FC_AngleToLength( _fDrivePos1,fDriveDiameter) )/fPoleWith )  ) ;  
      
		IF iUnwindStartTurns>=iUnwindOldTurns  AND  
             ABS( Driver.NcToPlc.SetVelo)<1  AND  VirMain.NcToPlc.ModuloActPos>=354 AND VirMain.NcToPlc.ModuloActPos<360    THEN  //   计算一次卷径
			_fDeltaDrivePos1:=ABS(Driver.NcToPlc.ActPos-_fDrivePos1);
			_fDeltaUwPos1:=ABS(Slave.NcToPlc.ActPos-_fUwPos1);
			_fDeltaDancerPos1:=fDanserDegree;
            DA1:=     f_Length2(Table:=Table,X:=_fDeltaDancerPos1)-f_Length2(Table:=Table,X:=_fDancerPos1) ;
			IF _fDeltaUwPos1<>0 THEN
          			 fDiameterCalculate:= ( FC_AngleToLength(_fDeltaDrivePos1,fDriveDiameter)- ( f_Length2(Table:=Table,X:=_fDeltaDancerPos1)-f_Length2(Table:=Table,X:=_fDancerPos1))  ) *360/ (PI*_fDeltaUwPos1) ;
		   	END_IF
            // fDiameterCalculate:= ( FC_AngleToLength(_fDeltaDrivePos1,fDriveDiameter)  ) *360/ (PI*_fDeltaUwPos1) ;
			_fDrivePos1:=Driver.NcToPlc.ActPos;		
			_fUwPos1:=Slave.NcToPlc.ActPos;
			_fDancerPos1:=fDanserDegree;
			iUnwindOldTurns:=10;
			fFlgCalculateOnce:=TRUE;
		END_IF
		
	END_IF

















(***********************************错误报警*********************************************)	
bAxisError:=      Slave.Status.Error OR  Master.Status.Error OR  TimerAxis.Status.Error ;
bFunBlokError:=fbGearDync.Error OR fbGearOut.Error OR fbHalt.Error OR fbJogUnwind.Error  ;
			
IF  bReset AND iTensionStep<>600  AND bError   THEN   //复位处理
    bError:=FALSE;
	iTensionStep:=630;
END_IF

(************************************  张力出错和取消的处理  ******************************************************)
Delay1(IN:=fDanserDegree>fDancerMaxPos AND bTensionOK , PT:=T#300MS , Q=> , ET=> );
bPosLimitError:=Delay1.Q;
Delay2(IN:=fDanserDegree<fDancerMinPos AND bTensionOK , PT:=T#300MS , Q=> , ET=> );
bNegLimitError:=Delay2.Q;
Delay3(IN:=( ABS(fActTorque -fSetTorque )>=10 OR  fDanserDegree> fDancerMaxPos+35 OR  fDanserDegree< fDancerMinPos-35)   AND   bTensionOK , PT:=T#300MS , Q=> , ET=> );
bTorqueError:=Delay3.Q;
Delay4(IN:=( iTensionStep=550 OR  iTensionStep=600 ) AND  Master.Status.NotMoving   AND (fDanserDegree>fDanceBlancePos+20  OR fDanserDegree<fDanceBlancePos-20)  AND ABS(fRatio2)>0.005 AND PidSwitch , PT:=T#5S , Q=> , ET=> );
bTenOKTimeError:=Delay4.Q;

Jog();
Motion();
TM_old:=TM;
*)

ACTION Jog:

CASE   iwindJog   OF
1: //收卷
    iFlgwind:=1;
	IF NOT bCcw THEN
	   fbJogUnwind.Jogbackwards :=TRUE;
		fbJogUnwind.JogForward:=FALSE;
	ELSE
		fbJogUnwind.JogForward:=TRUE;
		fbJogUnwind.Jogbackwards :=FALSE;
	END_IF
	iwindJog:=0;
2: //放卷
 iFlgwind:=2;
	IF NOT bCcw THEN
		fbJogUnwind.JogForward :=TRUE;
		fbJogUnwind.Jogbackwards:=FALSE;
	ELSE
		fbJogUnwind.Jogbackwards:=TRUE;
		fbJogUnwind.JogForward :=FALSE;
	END_IF
	iwindJog:=0;
3: //停止
     iFlgwind:=0;
	fbJogUnwind.Jogbackwards :=FALSE;
    fbJogUnwind.JogForward:=FALSE;
	iwindJog:=0;
END_CASE
END_ACTION

ACTION Motion:
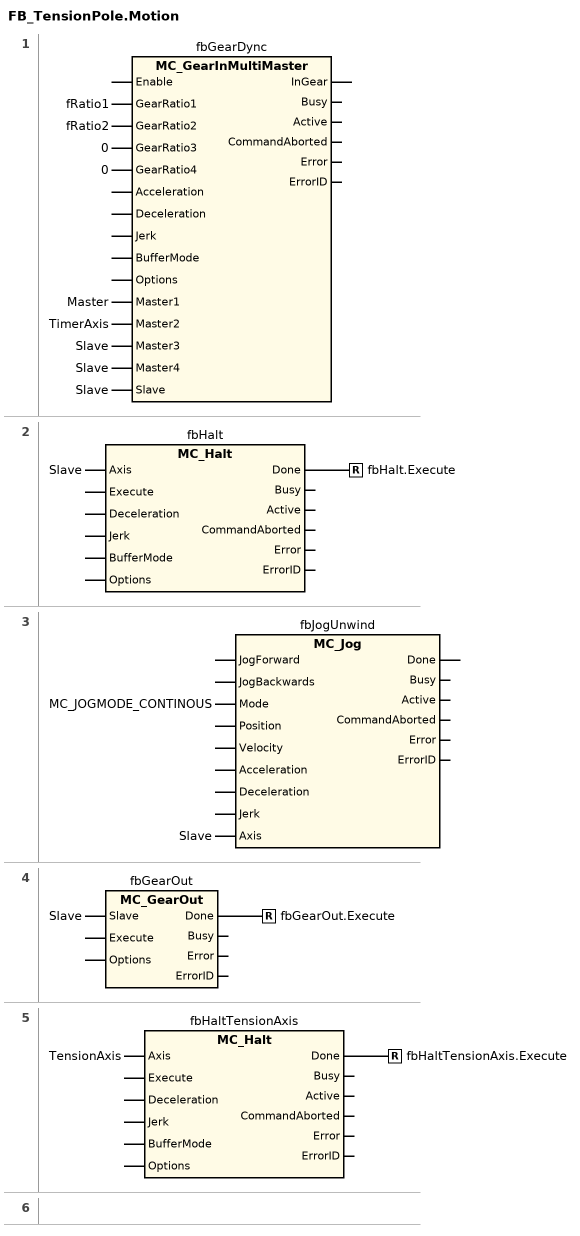
// NETWORK 1
fbGearDync(
    GearRatio1 := fRatio1,
    GearRatio2 := fRatio2,
    GearRatio3 := 0,
    GearRatio4 := 0,
    Master1 := Master,
    Master2 := TimerAxis,
    Master3 := Slave,
    Master4 := Slave,
    Slave := Slave); // MC_GearInMultiMaster

// NETWORK 2
fbHalt(Axis := Slave); // MC_Halt
fbHalt.Execute R= fbHalt.Done;

// NETWORK 3
fbJogUnwind(Mode := MC_JOGMODE_CONTINOUS, Axis := Slave); // MC_Jog

// NETWORK 4
fbGearOut(Slave := Slave); // MC_GearOut
fbGearOut.Execute R= fbGearOut.Done;

// NETWORK 5
fbHaltTensionAxis(Axis := TensionAxis); // MC_Halt
fbHaltTensionAxis.Execute R= fbHaltTensionAxis.Done;

// NETWORK 6
END_ACTION

ACTION Study:

rtStudy(CLK:=bStudyExecute, Q=> );
ftStudy(CLK:=bStudyExecute, Q=> );
IF rtStudy.Q THEN
	fbJogUnwind.Velocity:=2;
	bStudyFinish:=FALSE;
	bStudyExecute:=FALSE;
    studyStage:=1;
END_IF

IF ftStudy.Q THEN
	struckstudying:=FALSE;  
	bStudyFinish:=FALSE;
    studyStage:=40;
END_IF


CASE studyStage  OF 
	1:     //初始化
       	MEMSET(ADR(Table),0,SIZEOF(Table)); //  
		struckstudying:=TRUE;  
		structTime:=0;
		structPrinter:=1;  
		structAcc:=(fDancerMaxPos - fDancerMinPos)/100;  
	    studyStage := 2; 
   2:				
      IF fDanserDegree <= fDancerMinPos-1  THEN
		  iwindJog:=1;                         
          studyStage := 5; 
	  ELSE
	     iwindJog:=2;  
		 studyStage := 3; 
	  END_IF
   3:		  
      IF fDanserDegree < fDancerMinPos-1 THEN        
		  iwindJog:=1;                          
          studyStage := 5; 
	  END_IF	  	  
   5:	   
	IF Slave.Status.Moving AND Slave.Status.HasJob AND iwindJog=0 THEN 
		studyStage := 10;
	END_IF    
	10:
		ad_Set_test:=fDancerMinPos + structPrinter*structAcc;
		studyStage:=20;
	20:
(*
		IF 	ABS(fDanserDegree - ad_Set_test) < 0.2 THEN   
			structTime:=structTime+1;
	    ELSE
		    structTime:=0;
		END_IF
		IF structTime >= 3 THEN
			structTime:=0;
			structAxisPosPast := structAxisPosNow;  
			structAxisPosNow := Slave.NcToPlc.ActPos;   
			studyStage:=30;
		END_IF
*)
		IF 	fDanserDegree - ad_Set_test >0.1 THEN
			structAxisPosPast :=   structAxisPosNow;  
			structAxisPosNow :=  Slave.NcToPlc.ActPos;   
			studyStage:=30;
		END_IF

	30:
		IF structPrinter = 1 THEN
			Table[structPrinter - 1,1] := 0;
			Table[structPrinter - 1,2] := 0;
		 ELSE
			Table[structPrinter - 1,1] := ad_Set_test ; 
			Table[structPrinter - 1,2] := fStudyDiameter*PI/360*ABS((structAxisPosNow - structAxisPosPast)/gear) + Table[structPrinter - 2,2] ;
		END_IF
		structPrinter := structPrinter+1;
		
		IF structPrinter < 101  THEN
		 studyStage:=10;
		END_IF	
		 
		IF structPrinter = 101 OR ad_Set_test >= fDancerMaxPos THEN
            iwindJog:=3;
     		Table[0,1] := 0;//fDancerMinPos-10;
		    Table[0,2] := 0;//Table[1,2]-0.5;     
  
     		Table[100,1] := fDancerMaxPos+20;
		    Table[100,2] := Table[99,2]+0.5;     

			studyStage:=40;
		END_IF	
	40:
	        iwindJog:=3;
			bStudyExecute:=FALSE;
			bStudyFinish:=TRUE;
			struckstudying:=FALSE;
			studyStage:=0;
END_CASE

IF struckstudying AND  fDanserDegree>=fDancerMaxPos+4 AND  studyStage>=5 AND  Slave.Status.HasJob  THEN
	  iwindJog:=3;
	  studyStage:=0;
END_IF
END_ACTION

END_FUNCTION_BLOCK

// ---- POUs/BasicFunction/Motion/FB_Electric_CY.TcPOU
FUNCTION_BLOCK FB_Electric_CY
VAR_INPUT
    bServON   :BOOL;   
    bHome      :BOOL;   
    bReset      :BOOL;   
    bStop         :BOOL;   
    bJog_P         :BOOL;   
    bJog_N        :BOOL;   
    
   Pos_Start    :BOOL;   
   fTagetPos    :REAL;

   fVel:           REAL;
   fAcc        :REAL;  
   fDec        :REAL;  
   Delay_Time  :TIME;




END_VAR
VAR_OUTPUT
     bPowerOn       :BOOL;
     bHomed         :BOOL; 
     Pos_Done       :BOOL;   //定位完成
     Home_Alm      :BOOL;  //回零超时报警
     Pos_Alm         :BOOL; //定位超时报警

END_VAR

VAR_IN_OUT
    stJXCE   :ST_JXCE;

END_VAR




VAR





   rtHome    :Tc2_Standard.R_TRIG;
   tonHome   :Tc2_Standard.TON;
   rtPosStart    :Tc2_Standard.R_TRIG;

   tonPos   :Tc2_Standard.TON;
  tonPos2   :Tc2_Standard.TON;
  tonPos3   :Tc2_Standard.TON;
	bHomeIng: BOOL;
	Z_Pos: DINT;
	Z_Vel: UINT;
	Z_Acc: UINT;
	Z_Dec: UINT;
	bPosing: BOOL;


 //  iGoPos                :INT;   
//   iRealPos              :INT;
//   arrTagatPos         :ARRAY[1..5] OF REAL;  //目标点位



END_VAR



(****使能****)
   stJXCE.out_Control.9:= bServON;
   bPowerOn:=stJXCE.out_Control.9;
  
(****回零****)
rtHome(CLK:=bHome , Q=> );
 IF rtHome.Q AND  NOT  stJXCE.in_Status.8   THEN
    bHomeIng:=TRUE;
     bHomed:=FALSE;
END_IF

tonHome(IN:=bHomeIng , PT:=Delay_Time , Q=> , ET=> );
IF tonHome.Q THEN
    Home_Alm:=TRUE;
    bHomeIng:=FALSE;
END_IF

IF bReset AND Home_Alm THEN
     Home_Alm:=FALSE;
     bHomeIng:=FALSE;
    bHomed:=FALSE;
END_IF
stJXCE.out_Control.12:=bHomeIng;

IF bHomeIng AND stJXCE.in_Status.10 AND stJXCE.in_Status.11 THEN
    bHomed:=TRUE;
    bHomeIng:=FALSE;
END_IF

(********点动******)
stJXCE.out_Control.14:=bJog_P;
stJXCE.out_Control.13:=bJog_N;



(**********上使能后，速度，位置，加速度，减速度使能一直开启，定位默认为绝对模式**********)
stJXCE.out_Function.5:=stJXCE.out_Function.6:=stJXCE.out_Function.7:=stJXCE.out_Function.8:=stJXCE.in_Status.9;
IF stJXCE.in_Status.9 THEN
   stJXCE.out_Mode:=1;
	Z_Pos:=REAL_TO_DINT(fTagetPos*100);//HMI上位置单位为mm，电缸的位置单位为0.01mm
	stJXCE.out_Cmd_Pos:=Z_Pos;
	Z_Vel:=REAL_TO_UINT(fVel);//HMI上速度单位为mm/s，电缸的位置单位为mm/s
	Z_Acc:=REAL_TO_UINT(fAcc);//HMI上加速度单位为mm/s^2，电缸的加速度单位为mm/s^2
	Z_Dec:=REAL_TO_UINT(fDec);
	IF ABS( stJXCE.in_Act_Pos -stJXCE.out_Cmd_Pos) <=1 AND stJXCE.in_Status.11      THEN
		Pos_Done:=TRUE;
	ELSE
		Pos_Done:=FALSE;
	END_IF
END_IF


rtPosStart(CLK:=Pos_Start  , Q=> );
IF rtPosStart.Q THEN
	IF    stJXCE.in_Status.9  AND  stJXCE.in_Status.10  AND stJXCE.out_Start=0   THEN
		 stJXCE.out_Cmd_Pos:=Z_Pos;
  	    stJXCE.out_Cmd_Vel:=Z_Vel;
		 stJXCE.out_Cmd_Acc:=Z_Acc;
		 stJXCE.out_Cmd_Dec:=Z_Dec;
		 stJXCE.out_Start:=1;
		  bPosing:=TRUE;
		  Pos_Alm:=FALSE;
	END_IF
	
	IF  NOT  stJXCE.in_Status.9  OR NOT  stJXCE.in_Status.10 THEN
	       Pos_Alm:=TRUE;
	END_IF

END_IF

tonPos(IN:=stJXCE.out_Start<>0 , PT:=T#500MS , Q=> , ET=> );
IF tonPos.Q THEN
    stJXCE.out_Start:=0;
END_IF 

tonPos2(IN:=bPosing , PT:=Delay_Time , Q=> , ET=> );
IF tonPos2.Q THEN
		  bPosing:=FALSE;
		  Pos_Alm:=TRUE;
END_IF


IF bReset AND Pos_Alm THEN
		  bPosing:=FALSE;
		  Pos_Alm:=FALSE;
END_IF

tonPos3(IN:=bPosing , PT:=T#100MS , Q=> , ET=> );
IF tonPos3.Q  AND  stJXCE.in_Status.11   THEN
     bPosing:=FALSE;
    stJXCE.out_Start:=0;
END_IF
















(***复位*)
//stJXCE.out_Control.11:=( bReset AND stJXCE.in_Latest_Alm<>0 )   OR  bStop ;

stJXCE.out_Control.11:=( bReset AND stJXCE.in_Latest_Alm<>0 )   OR  bStop ;

END_FUNCTION_BLOCK

// ---- POUs/BasicFunction/User1/FB_DataXML_Old.TcPOU
FUNCTION_BLOCK FB_DataXML_Old
VAR_INPUT
    	bSave:BOOL;
	    bRead:BOOL;

		
END_VAR
VAR_OUTPUT
    	bSaveParDone      :BOOL;
	    bReadParDone     :BOOL;
		bError                     :BOOL;   
END_VAR

VAR


	iDataSetp: INT;
	TON10:Tc2_Standard.TON;
	I1: INT;
	rt100:Tc2_Standard.R_TRIG;
	rt101:Tc2_Standard.R_TRIG;
	bExecute1: BOOL;
	bExecute2: BOOL;


	bSaveTemp: BOOL;
	bReadTemp: BOOL;

 fbXmlSrvWrite         : FB_XmlSrvWrite;
// fbXmlSrvWrite         : FB_SrvWrite;
   bExecuteW1             : BOOL;
   sFilePathPar_W       : T_MaxString ;

  // value2                : ST_MYSTRUCT;
fbXmlSrvRead   : FB_XmlSrvRead;
//fbXmlSrvRead   : FB_SrvRead;
   bExecuteR          : BOOL;
   sFilePathPar_R      : T_MaxString ;
   sXPathR             : T_MaxString;
	AA: INT;
	BB: INT;












	handleTemp: UDINT;
	//rtResetSaveDone: R_TRIG;
	//rtResetReadDone: R_TRIG;
END_VAR


M_WriteOrRead();

ACTION M_WriteOrRead:
bError:=fbXmlSrvWrite.bError OR fbXmlSrvRead.bError;

rt100(CLK:=bSave , Q=> );//保存参数
rt101(CLK:=bRead , Q=> );//读取参数

IF rt100.Q THEN  //保存参数
	iDataSetp:=100;
	TON10.IN:=FALSE;
	I1:=1;
	bExecute1:=FALSE;
	bExecute2:=FALSE;
	bSave:=FALSE;
	bRead:=FALSE;
    bSaveTemp:=TRUE;
	bReadTemp:=FALSE;
	bSaveParDone:=FALSE;
END_IF

IF rt101.Q THEN  //读取参数
	iDataSetp:=100;
	TON10.IN:=FALSE;
	I1:=1;
	bExecute1:=FALSE;
	bExecute2:=FALSE;	
	bSave:=FALSE;
	bRead:=FALSE;
    bReadTemp:=TRUE;
    bSaveTemp:=FALSE;
	bReadParDone:=FALSE;
END_IF

TON10(IN:= , PT:=T#200MS , Q=> , ET=> );


(*
rtResetSaveDone(CLK:=NOT bSave  AND  bSaveParDone  , Q=> );
IF  rtResetSaveDone.Q THEN
	bSaveParDone:=FALSE;
END_IF
rtResetReadDone(CLK:=NOT bRead  AND  bReadParDone  , Q=> );
IF  rtResetReadDone.Q THEN
	bReadParDone:=FALSE;
END_IF
*)



CASE  iDataSetp OF 
	
 100:
				CASE I1 OF 
				  1://轴参数
					sFilePathPar_W  := 'C:\P1XML\P1arrAxisPar.xml';
					fbXmlSrvWrite.pSymAddr:=ADR(arrAxisPar);
					fbXmlSrvWrite.cbSymSize:=SIZEOF(arrAxisPar);   

					sFilePathPar_R  := 'C:\P1XML\P1arrAxisPar.xml';
					fbXmlSrvRead.pSymAddr:=ADR(arrAxisPar);
					fbXmlSrvRead.cbSymSize:=SIZEOF(arrAxisPar);   
     
				  2://ProductPar
		  		    sFilePathPar_W  := 'C:\P1XML\P1ProductPar.xml';
					fbXmlSrvWrite.pSymAddr:=ADR(ProductPar);
					fbXmlSrvWrite.cbSymSize:=SIZEOF(ProductPar);     

					sFilePathPar_R  :=  'C:\P1XML\P1ProductPar.xml';
					fbXmlSrvRead.pSymAddr:=ADR(ProductPar);
					fbXmlSrvRead.cbSymSize:=SIZEOF(ProductPar);   
(*					
				  3://Name
		  		     sFilePathPar_W  := 'C:\P1XML\P1Name.xml';
					fbXmlSrvWrite.pSymAddr:=ADR(NameNo);
					fbXmlSrvWrite.cbSymSize:=SIZEOF(NameNo);     

					sFilePathPar_R  := 'C:\P1XML\P1Name.xml';
					fbXmlSrvRead.pSymAddr:=ADR(NameNo);
					fbXmlSrvRead.cbSymSize:=SIZEOF(NameNo);   

				  4://Data
		  		    sFilePathPar_W  := 'C:\P1XML\P1Data.xml';
					fbXmlSrvWrite.pSymAddr:=ADR(PoleData);
					fbXmlSrvWrite.cbSymSize:=SIZEOF(PoleData);     

					sFilePathPar_R  := 'C:\P1XML\P1Data.xml';
					fbXmlSrvRead.pSymAddr:=ADR(PoleData);
					fbXmlSrvRead.cbSymSize:=SIZEOF(PoleData);   

				  5: //P2M3_Par 
		  		    sFilePathPar_W  := 'C:\XML\P2M3_Par.xml';
					fbXmlSrvWrite.pSymAddr:=ADR(P2M3_Par);
					fbXmlSrvWrite.cbSymSize:=SIZEOF(P2M3_Par);     

					sFilePathPar_R  := 'C:\XML\P2M3_Par.xml';
					fbXmlSrvRead.pSymAddr:=ADR(P2M3_Par);
					fbXmlSrvRead.cbSymSize:=SIZEOF(P2M3_Par);   		
*)					
				END_CASE
        IF  bSaveTemp THEN
              handleTemp:=fbXmlSrvWrite.handle;
   	          iDataSetp:=200;
       END_IF
        IF  bReadTemp THEN
              handleTemp:=fbXmlSrvRead.handle;
   	          iDataSetp:=300;
       END_IF

	200:	//保存数据
		bExecute1:=TRUE;
        iDataSetp:=210;
	210:	
       IF  NOT fbXmlSrvWrite.bError  AND NOT fbXmlSrvWrite.bBusy AND handleTemp<>fbXmlSrvWrite.handle  THEN
             iDataSetp:=500;
      END_IF

	300:	//读取参数
		bExecute2:=TRUE;
        iDataSetp:=310;
	310:	
       IF  NOT fbXmlSrvRead.bError  AND NOT fbXmlSrvRead.bBusy AND handleTemp<>fbXmlSrvRead.handle  THEN
             iDataSetp:=500;
      END_IF


	500://继续写下个文件
	  IF I1>=1 AND I1<3 THEN
		 I1:=I1+1; 
		 iDataSetp:=100; 
		 bExecute1:=FALSE; 
		 bExecute2:=FALSE; 
	  ELSIF I1>=3 THEN
          IF  bSaveTemp THEN
               bSaveParDone:=TRUE;
         END_IF

          IF  bReadTemp THEN
               bReadParDone:=TRUE;
         END_IF

		  bReadTemp:=FALSE;
          bSaveTemp:=FALSE;

	   	 iDataSetp:=666;   
	  END_IF
END_CASE



AA:=BB;

fbXmlSrvWrite(
   nMode           := XMLSRV_ADDMISSING,
   pSymAddr        :=,//ADR(Value1)
   cbSymSize       := ,//SIZEOF(Value1)
   sFilePath       := sFilePathPar_W,
   sXPath	       := '/dataentry/value',
   bExecute        := bExecute1
);
fbXmlSrvWrite.nErrId;


fbXmlSrvRead(
   pSymAddr       := ,
   cbSymSize      := ,
   sFilePath      := sFilePathPar_R,
   sXPath	         := '/dataentry/value',
   bExecute       := bExecute2
);
END_ACTION

END_FUNCTION_BLOCK

// ---- POUs/BasicFunction/XFC/FB_EL1259_IN.TcPOU
FUNCTION_BLOCK FB_EL1259_IN  //单次触发

(*本FB适用于EL1258和EL1259的输入通道*)

VAR
	aIE_Time  AT%I* :   UDINT;
  	aIE_State AT%I*:  BOOL;
	nEventsInInputBuffer AT%I*: USINT;
	nNoOfInputEvents AT %I*:USINT;
	bInputState AT%I* :  BOOL ;
	bInputBufferReset AT %Q*:BOOL;


END_VAR
VAR_INPUT
	cmdInputBufferReset: BOOL;
END_VAR


bInputBufferReset:=cmdInputBufferReset;

END_FUNCTION_BLOCK

// ---- POUs/BasicFunction/XFC/FB_TouchProbe_Ear.TcPOU
FUNCTION_BLOCK  FB_TouchProbe_Ear   //负极极而XFC

VAR_INPUT
   	aIE_Time   :  UDINT;  (*上升沿或者下降沿的Event 时间*)
  	aIE_State   : BOOL;	(*State为TRUE，表示Event为上升沿，为False，表示Event是下降沿*)
	nNoOfInputEvents :USINT;			(*本周期发生的Event数量*)
	bInputState :  BOOL ;				(*当前输入最后一次更新状态*)
END_VAR

VAR_IN_OUT
	bXfcOk :BOOL;
 	Axis			:	 Axis_Ref ;
	TriggerInput	:	XFC_TRIGGER_REF;
END_VAR

VAR_OUTPUT
	bFunBlockError :BOOL;
	RecordedPos	: LREAL;(*锁存结果*)
END_VAR

VAR
	XFC_TouchProbe:  XFC_TouchProbe;// XFCFB
	XFC_TriggerInput: XFC_TRIGGER_REF;
	R_TRGIG: R_TRIG;
	rTrigClear: F_TRIG;
	rTrigStart: R_TRIG;
	
	fTrigStart: F_TRIG;	
	fPosIo: LREAL;
	fPosDelta: LREAL;
	arrfPosDelta: ARRAY[1..500] OF LREAL;
	fPos1: LREAL;
	K1 :DINT:=1;
	bClear: BOOL;
	iSetp: INT;
    iXFCStatus: INT;
	uI1: UINT;
	b2: BOOL;
	aIE_StateTemp: BOOL;
	bIoRecordDataOk: BOOL;
	//RecordedPos1: LREAL;
	DD1: INT;
	//AA1: BOOL;
	//AA2: BOOL;
	//AA3: INT;
	bAxisMoving: BOOL;
	fPos3: LREAL;
	RecordedPositionXFC: LREAL;
	K2: INT;
	K3: DINT;
	K4: DINT;
	MB3: BOOL;
END_VAR

XFC_TriggerInput:=TriggerInput;  //配置参数传递


rTrigStart(CLK:= XFC_TriggerInput.Signal , Q=> ); // nNoOfInputEvents>0	
fTrigStart(CLK:= XFC_TriggerInput.Signal , Q=> ); // nNoOfInputEvents>0

bAxisMoving:= Axis.Status.Moving ;

IF fTrigStart.Q AND bAxisMoving THEN    //下降沿取值
    fPosIo:=Axis.NcToPlc.ModuloActPos; //IO记录位置
	bIoRecordDataOk:=TRUE;
END_IF

//确保XFC 和IO数据传递过来
IF bIoRecordDataOk AND iXFCStatus=1  THEN
	fPosDelta:=RecordedPositionXFC-fPosIo;	 //差值	
	arrfPosDelta[K1]:=fPosDelta;	//偏差值记录
 
	 K1:=K1+1;
    bIoRecordDataOk:=FALSE;
	iXFCStatus:=3;
END_IF

IF K1>=500 THEN 
	K1:=1;
END_IF

rTrigClear(CLK:=bClear , Q=> );   
IF rTrigClear.Q THEN					(*清空记录*)
	MEMSET(ADR(arrfPosDelta),0,SIZEOF(arrfPosDelta)); 
    K1:=K4:=K3:=1;
END_IF

(*****XFC******)
R_TRGIG(CLK:=nNoOfInputEvents>=1 AND bAxisMoving , Q=> );
IF R_TRGIG.Q THEN
	bXfcOk:=FALSE;
	RecordedPositionXFC:=0;
    K2:=K2+1;
	iSetP:=10;
END_IF


IF aIE_State THEN
  XFC_TriggerInput.Edge:=Tc2_MC2.RisingEdge;
  XFC_TriggerInput.TimestampRisingEdge := aIE_Time;  //识别时间输入 上升沿
   MB3:=TRUE;
ELSE
    XFC_TriggerInput.Edge:=Tc2_MC2.FallingEdge;
	XFC_TriggerInput.TimestampFallingEdge := aIE_Time;  //识别时间输入  下降沿
   MB3:=FALSE;
END_IF

IF  nNoOfInputEvents=0 THEN
	 RETURN;
END_IF

IF iSetp=10 THEN
	bXfcOk:=FALSE;
    K4:=K4+1;
	XFC_TouchProbe(
		Axis:=                     Axis , 
		TriggerInput:=         XFC_TriggerInput, 
		Execute:=                TRUE, 
		WindowOnly:=        FALSE , 
		FirstPosition:=          0 , 
		LastPosition:=          0, 
		Options:= , 
		Done=> , 
		Busy=> , 
		Error=> , 
		ErrorID=> , 
		RecordedPosition=> );//XFC_TouchProbe.RecordedPosition
	   XFC_TouchProbe.Done;		
	   XFC_TouchProbe.Busy;		
	  XFC_TouchProbe.Error;		
	  XFC_TouchProbe.ErrorID;	 

    IF XFC_TriggerInput.Edge=FallingEdge THEN
      RecordedPositionXFC:=XFC_TouchProbe.RecordedPosition;
       RecordedPos:=RecordedPositionXFC;
          K3:=K3+1;
       	bXfcOk:=TRUE;
       iXFCStatus:=1; 
    ELSE 
       iXFCStatus:=2; 
   END_IF
     iSetp:=88 ;
END_IF



(*
IF  nNoOfInputEvents=0 THEN
	 RETURN;
END_IF
*)

END_FUNCTION_BLOCK

// ---- POUs/BasicFunction/Data/CS_Data_Test.TcPOU
FUNCTION_BLOCK CS_Data_Test
VAR_INPUT
END_VAR
VAR_OUTPUT
END_VAR
VAR
	//tDataSave:TON;
	//fbSaveData:FB_WritePersistentData;
	//fbXMLWrite:FB_XMLSrvWrite;
	//bWriteXml: BOOL;
	
	fbFileOpen_w:fb_fileopen;
	//fbFileOpen_r:fb_fileopen;
	fbFileWrite:fb_filewrite;
	fbFileRead:FB_FileRead;
	fbFileClose_w:fb_FileClose;
	//fbFileClose_r:fb_FileClose;
	HFILE:UINT;
	//HFILE_R:UINT;
	//bFileOpen_w:BOOL;
	//bFileOpen_r:BOOL;
	//bFileWrite:BOOL;
	//bFileClose_w:BOOL;
	//bFileClose_r:BOOL;
	//bFileRead:BOOL;
	bSave:BOOL;
	bRead:BOOL;
//	tFileOper_Save:TON;
	//tFileOper_Read:TON;
	iDataSetp: INT;
	TON10:Tc2_Standard.TON;
	bExecute: BOOL;
	I1: INT;
	rt100:Tc2_Standard.R_TRIG;
	rt101:Tc2_Standard.R_TRIG;
	bExecute1: BOOL;
	bExecute2: BOOL;
	bExecute3: BOOL;	

	bSaveTemp: BOOL;
	bReadTemp: BOOL;
	bReadDataOk: BOOL;
END_VAR





M_WriteOrRead();

ACTION M_WriteOrRead:



rt100(CLK:=bSave , Q=> );//保存参数
rt101(CLK:=bRead , Q=> );//读取参数

IF rt100.Q THEN
	iDataSetp:=100;
	TON10.IN:=FALSE;
	I1:=1;
	bExecute1:=FALSE;
	bExecute2:=FALSE;	
	bExecute3:=FALSE;	
	bSave:=FALSE;
	bRead:=FALSE;
    bSaveTemp:=TRUE;
	bReadTemp:=FALSE;
END_IF

IF rt101.Q THEN
	iDataSetp:=100;
	TON10.IN:=FALSE;
	I1:=1;
	bExecute1:=FALSE;
	bExecute2:=FALSE;	
	bExecute3:=FALSE;	
	bSave:=FALSE;
	bRead:=FALSE;
    bReadTemp:=TRUE;
    bSaveTemp:=FALSE;
END_IF

TON10(IN:= , PT:=T#200MS , Q=> , ET=> );
//保存配方	
CASE  iDataSetp OF 
	
	100:	//参数给定
	   
	   IF bSaveTemp THEN
	     fbFileOpen_w.nMode:=FOPEN_MODEWRITE OR FOPEN_MODEBINARY;
	   END_IF
	   IF bReadTemp THEN
	     fbFileOpen_w.nMode:=FOPEN_MODEREAD OR  FOPEN_MODEBINARY;
	   END_IF
	  iDataSetp:=101;
	101:

	  CASE I1 OF 
		1:
		 fbFileWrite.pWriteBuff:=ADR(gstM1Par);
		 fbFileWrite.cbWriteLen:=SIZEOF(gstM1Par);
		 fbFileRead.pReadBuff:=ADR(gstM1Par1);
		 fbFileRead.cbReadLen:=SIZEOF(gstM1Par1);
		 fbFileOpen_w.sPathName:='C:\P2Data\M1.csv';//='C:\P2Data\M1.bin';

	  END_CASE
	  iDataSetp:=200;
	
	200:	//打开文件
		bExecute1:=TRUE;
		TON10.IN:=TRUE;
	  IF TON10.Q THEN
		 bExecute1:=FALSE; 
		 TON10.IN:=FALSE;
		 iDataSetp:=300; 
	  END_IF
	
	300:	//读写文件
		bExecute2:=TRUE;
		TON10.IN:=TRUE;
	  IF TON10.Q THEN
		  bExecute2:=FALSE; 
		  TON10.IN:=FALSE;
		 iDataSetp:=400; 
	  END_IF
	
	400:	//关闭文件
		bExecute3:=TRUE;
		TON10.IN:=TRUE;
	  IF TON10.Q THEN
		  bExecute3:=FALSE; 
		  TON10.IN:=FALSE;
		  iDataSetp:=500; 
	  END_IF
	
	500://继续写下个文件
	  IF I1>=1 AND I1<5 THEN
		 I1:=I1+1; 
		 TON10.IN:=FALSE;
		 iDataSetp:=100; 
		 bExecute1:=FALSE; 
		 bExecute2:=FALSE; 
		 bExecute3:=FALSE; 
	  ELSIF I1>=5 THEN
		  bReadTemp:=FALSE;
          bSaveTemp:=FALSE;
		 iDataSetp:=666;   
	  END_IF
END_CASE


IF bReadDataOk THEN
   gstM1Par:=gstM1Par1;
   gstM2Par:=gstM2Par1;
   gstM3Par:=gstM3Par1;
   gstM4Par:=gstM4Par1;	
   gstM5Par:=gstM5Par1;
   bReadDataOk:=FALSE;
END_IF










   	fbFileOpen_w(
	sNetId:= , 
	sPathName:= , //C:\P2Data
	nMode:=   , 
	ePath:=PATH_GENERIC , 
	bExecute:=bExecute1 , 
	tTimeout:=T#3S , 
	bBusy=> , 
	bError=> , 
	nErrId=> , 
	hFile=>hfile );


	fbFileWrite(
	sNetId:= , 
	hFile:= hFile, 
	pWriteBuff:= , 
	cbWriteLen:= , 
	bExecute:=bExecute2 AND bSaveTemp, 
	tTimeout:=T#3S , 
	bBusy=> , 
	bError=> , 
	nErrId=> , 
	cbWrite=> );



	fbFileRead(
	sNetId:= , 
	hFile:=hFile , 
	pReadBuff:= , 
	cbReadLen:= , 
	bExecute:= bExecute2 AND bReadTemp, 
	tTimeout:= T#3S, 
	bBusy=> , 
	bError=> , 
	nErrId=> , 
	cbRead=> , 
	bEOF=> );


	fbFileClose_w(
	sNetId:= , 
	hFile:= hFile, 
	bExecute:= bExecute3, 
	tTimeout:=T#3S , 
	bBusy=> , 
	bError=> , 
	nErrId=> );
END_ACTION

END_FUNCTION_BLOCK

// ---- POUs/BasicFunction/MES/CS_CcdTcp.TcPOU
FUNCTION_BLOCK PUBLIC CS_CcdTcp
VAR_INPUT
END_VAR
VAR_OUTPUT
END_VAR
VAR_IN_OUT
   iCcd2:ST_CCDCom;
   Data:STCcdData;
END_VAR


VAR
	ccdDataSend:STCcdDataSend;
	
	fbTcpCon:FB_SocketConnect;
	fbTcpSend:FB_SocketSend;
	fbTcpRec:FB_SocketReceive;
	fbTcpClose: FB_SocketClose;
	bConnect: BOOL;
	bClose: BOOL;
	hTcpSock: T_HSOCKET;
	//aTcpSend:ARRAY[1..10] OF BYTE;
	//aTcpReceive:ARRAY[1..10] OF BYTE;	
	StrSend:STRING;
	StrReceive:STRING;
	fbUdpCreate:FB_SocketUdpCreate;
	hUdp: T_HSOCKET;
	bCreate: BOOL;
	port: UDINT:=9004;
	bSendTcp: BOOL;
	bReceiveTcp: BOOL;
	fbSwingHalt2: MC_Halt;



END_VAR




	Config();
	
	M_SendReceive();


	
	

	
	
	
	

	
	
	
	
	
	
	
	
	
	
	
	
	
	
	
	
	
(*	
   fbUdpCreate(
	sSrvNetId:= , 
	sLocalHost:= , 
	nLocalPort:= port, 
	bExecute:=bCreate , 
	tTimeout:= , 
	bBusy=> , 
	bError=> , 
	nErrId=> , 
	hSocket=> hUdp);
	
	
	*)

ACTION Config:



  IF iCcd2.bComOpen THEN
	 bConnect:=TRUE;	
	 bClose:=FALSE;
	 iCcd2.bComOpen:=FALSE;
  END_IF
  
   IF iCcd2.bComClose THEN
	 bConnect:=FALSE;	
	 bClose:=TRUE;
	 iCcd2.bComClose:=FALSE;
  END_IF 
  
  
  
fbTcpCon(
	sSrvNetId:= ''   ,          //       (*'169.254.46.193.1.1'*) , 
	sRemoteHost:='192.168.2.11'     , 
	nRemotePort:= 2020, 
	bExecute:=bConnect , 
	tTimeout:= , 
	bBusy=> , 
	bError=> , 
	nErrId=> , 
	hSocket=>hTcpSock );
	
fbTcpClose(
	sSrvNetId:= ''   , 
	hSocket:=hTcpSock , 
	bExecute:=bClose , 
	tTimeout:=T#5S , 
	bBusy=> , 
	bError=> , 
	nErrId=> );


IF fbTcpCon.bBusy THEN
	bConnect:=FALSE;
END_IF

IF fbTcpClose.bBusy THEN
   bClose:=FALSE;
END_IF
END_ACTION

ACTION M_SendReceive:


  IF iCcd2.bSend THEN
	 bSendTcp:=TRUE;
	 iCcd2.bDone:=FALSE;
	 iCcd2.bError:=FALSE;
	 //iCcd2.strReceive:='';
    MEMSET(ADR(ccdDataSend.strBetryName),0,SIZEOF(ccdDataSend.strBetryName));
	MEMSET(ADR(ccdDataSend.strCode),0,SIZEOF(ccdDataSend.strCode));
	MEMSET(ADR(ccdDataSend.strShortData),0,SIZEOF(ccdDataSend.strShortData));
	MEMSET(ADR(ccdDataSend.strHotPress),0,SIZEOF(ccdDataSend.strHotPress));
    STRING_TO_UTF8(pDstUTF8:=ADR(ccdDataSend.strBetryName) , pSrcSTRING:=ADR(Data.strBetryName) , nDstSize:=INT_TO_UINT( LEN(STR:=Data.strBetryName )+1) );
    STRING_TO_UTF8(pDstUTF8:=ADR(ccdDataSend.strCode) , pSrcSTRING:=ADR(Data.strCode) , nDstSize:=INT_TO_UINT( LEN(STR:=Data.strCode )+1) ); 
    STRING_TO_UTF8(pDstUTF8:=ADR(ccdDataSend.strShortData) , pSrcSTRING:=ADR(Data.strShortData) , nDstSize:=INT_TO_UINT( LEN(STR:=Data.strShortData )+1) );
	STRING_TO_UTF8(pDstUTF8:=ADR(ccdDataSend.strHotPress) , pSrcSTRING:=ADR(Data.strHotPress) , nDstSize:=INT_TO_UINT( LEN(STR:=Data.strHotPress )+1) );
    iCcd2.bSend:=FALSE;
END_IF
	 


fbTcpSend(
		sSrvNetId:= , 
		hSocket:=hTcpSock , 
		cbLen:=SIZEOF(ccdDataSend), 
		pSrc:= ADR(ccdDataSend), 
		bExecute:= bSendTcp, 
		tTimeout:= T#2S , 
		bBusy=> , 
		bError=> , 
		nErrId=> );
	IF bSendTcp AND fbTcpSend.bBusy THEN
		bSendTcp:=FALSE;
	END_IF
	
	
bReceiveTcp:=NOT bReceiveTcp;
	
fbTcpRec(
	sSrvNetId:= , 
	hSocket:= hTcpSock, 
	cbLen:=SIZEOF(StrReceive) , 
	pDest:=ADR(StrReceive) , 
	bExecute:=bReceiveTcp , 
	tTimeout:= T#5S, 
	bBusy=> , 
	bError=> , 
	nErrId=> , 
	nRecBytes=> );

IF LEN(STR:=StrReceive )>=10 THEN
  iCcd2.strReceive:=StrReceive;
  StrReceive:='';
 // iCcd2.bDone:=TRUE;
END_IF


//IF LEN(STR:=StrReceive )=0 THEN
END_ACTION

END_FUNCTION_BLOCK
